// TIA Portal V16 export
// export: Created 2022-01-12T14:34:26.780226Z, ExportSetting WithDefaults, DisplayName Totally Integrated Automation Portal, DisplayVersion V16 Update 4, DisplayName TIA Portal Version Control Interface, DisplayVersion V16 Update 2, DisplayName TIA Portal Openness, DisplayVersion V16 Update 4, DisplayName STEP 7 Professional, DisplayVersion V16 Update 4, DisplayName STEP 7 Safety, DisplayVersion V16, DisplayName WinCC Professional, DisplayVersion V16 Update 4
TYPE "typKrokRecepturyStacjiMycia"
// stored: IsFailsafeCompliant false
   STRUCT
      nazwaKroku : WString[33] := WSTRING#'nazwa receptury';   // nazwa kroku
      PM : Array[0..30] of Real;
   END_STRUCT;
   // // PM[1] : krokAktywny
   // // PM[2] : wydajnośćMycia
   // // PM[3] : czasOczekiwaniaNaZasilanie
   // // PM[4] : CzasOczekiwaniaNaPowrót
   // // PM[5] : ObjętośćPłukania
   // // PM[6] : CzasMycia
   // // PM[7] : CzasOdsączania
   // // PM[8] : Objetość WypełnieniaDoGruszki
   // // PM[9] : CzasOpóżnieniaUruchomieniaPompyCIP
   // // PM[10] : StężeniaMinimalne
   // // PM[11] : StężenieDozowania
   // // PM[12] : StężeniePłukania
   // // PM[13] : TemperaturaProcesu
   // // PM[14] : TemperaturaPłukania
   // // PM[15] : HisterezaStężeniaDoRozpoczęciaOdliczania
   // // PM[16] : RóznicaTemperaturDoRozpoczęciaOdliczania
   // // PM[17] : WspółczynnikKompensacji
   // // PM[18] : TemperaturaOdniesieniaKompensacji
   // // PM[19] : MaksymalnyCzasOperacji
   // // PM[20] : CzasDozowaniaChemii
   // // PM[21] : SprawdzanieCzujników
   // // PM[22] : KompensacjaTemperaturowa
   // // PM[23] : MycieTanku
   // // PM[24] : CIPsp201 optymalizacja objetosci
   // // PM[25] : Cipsp202 optymalizacja stezen
   // // PM[26] : czas załączenia pompki chemii
   // // PM[27] : czas wyłączenia pompki chemii
END_TYPE
